{attribute 'GeneratedUsingTerminal: ELX9560-0000-0016'}
{attribute addProperty BoxType "ELX9560-0000-0016"}
{attribute addProperty Id "Power_OKAT %I*BOOL1"}
{attribute addProperty CRC "1151167157"}
{attribute addProperty Size "1"}
TYPE Status_Uex_449D6AB5 EXTENDS InputBase_8311D824 :
STRUCT
	{attribute addProperty Name "Power_OK"}
	Power_OK AT %I* : BOOL;
END_STRUCT
END_TYPE

(* stored: Version 1.2.0.0, ProductVersion 3.1.4024.11
   DUT Status_Uex_449D6AB5: Id {055c7720-acff-4001-b50a-5def96a65c08} *)
